Staubli VAL3: RecordAddon.dtx

jointRx jJoint[3]
  [0] = {j1=-31.315744, j3=72.801072, j5=40.352904}
  [1] = {j1=-13.5, j3=72.801072, j5=40.352904}
  [2] = {j1=17.815744, j3=72.801072, j5=40.352904}
mdesc mNomSpeed
mdesc mSpeed = {accel=20, decel=20, tmax=100, blend=cartesian, leave=1, reach=1}
